{attribute 'qualified_only'}
VAR_GLOBAL
	flSS1				: FB_BaseFlag;
	flSTO				: FB_BaseFlag;
	
END_VAR

(* stored: Version 1.1.0.1
   GVL GVL_MCSafety: Id {408e1c6e-7663-05c5-1c01-34065daabb61} *)
